FUNCTION INTERNAL F_IsPackedRepeatedField : BOOL
VAR_INPUT
    nTag : UDINT;
END_VAR


F_IsPackedRepeatedField := F_GetTagWireType(nTag) = E_WireType.LengthDelimited;

END_FUNCTION

(* stored: Version 1.1.0.1
   POU F_IsPackedRepeatedField: Id {9ddab4bb-5e29-4edf-8769-6b2defee71d6}, SpecialFunc None *)
